FUNCTION TryConvert_BYTE_TO_UDINT : BOOL
VAR_INPUT
	in : BYTE;
	out : REFERENCE TO UDINT;
END_VAR

out := BYTE_TO_UDINT(in);
TryConvert_BYTE_TO_UDINT := TRUE;

END_FUNCTION

(* stored: Version 1.1.0.1, ProductVersion 3.1.4024.12
   POU TryConvert_BYTE_TO_UDINT: Id {180cc63d-9ab8-440a-adb2-5595a5053c77}, SpecialFunc None *)
